TYPE timeDry :
STRUCT
	dia: STRING;
	hora: string;
END_STRUCT
END_TYPE

(* stored: Version 1.1.0.1, ProductVersion 3.1.4024.12
   DUT timeDry: Id {01ecff7d-8417-4241-acd2-9f0dfa4d52ee} *)
